FUNCTION_BLOCK OR_8 (* FB to calculate bitwise boolean OR (generic FB) *)
  PACKAGE iec61131::arithmetic;
  {SET_ATTRIBUTE(eclipse4diac::core::GenericClassName, 'GEN_OR')}
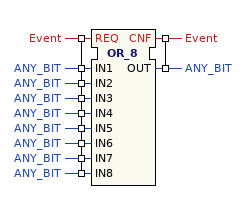
  EVENT_INPUT
    REQ WITH IN1, IN2, IN3, IN4, IN5, IN6, IN7, IN8; (* Normal Execution Request *)
  END_EVENT
  EVENT_OUTPUT
    CNF WITH OUT; (* Execution Confirmation *)
  END_EVENT
  VAR_INPUT
    IN1 : ANY_BIT; (* OR input 1 *)
    IN2 : ANY_BIT; (* OR input 2 *)
    IN3 : ANY_BIT; (* OR input 3 *)
    IN4 : ANY_BIT; (* OR input 4 *)
    IN5 : ANY_BIT; (* OR input 5 *)
    IN6 : ANY_BIT; (* OR input 6 *)
    IN7 : ANY_BIT; (* OR input 7 *)
    IN8 : ANY_BIT; (* OR input 8 *)
  END_VAR
  VAR_OUTPUT
    OUT : ANY_BIT; (* OR result *)
  END_VAR
END_FUNCTION_BLOCK
